// TIA Portal V19 export
DATA_BLOCK "Coilcar"   // DB112
// stored: InstanceOfName Coilcar_FB, InstanceOfType FB
"Coilcar_FB"
   // VAR_INPUT
   //    AreaInterface : "AreaInterface";
   //    ZSI : "udt_ZoneSafetyInterface";
   //    DSI : Struct
   //       Move : "udt_DeviceSafetyInterface";
   //       LIft : "udt_DeviceSafetyInterface";
   //    END_STRUCT;
   //    Drive : "TAx_DriveInterface";
   //    HW_ID_TEL1 : HW_SUBMODULE;
   //    DataIn : Struct
   //       Supports_Ls_FixPoleLeft_Plugged : Bool;
   //       Supports_Ls_FixPoleRight_Plugged : Bool;
   //       Supports_Ls_MobilePoleLeft_Plugged : Bool;
   //       Supports_Ls_MobilePoleRight_Plugged : Bool;
   //       Move_Ls_Outline : Bool;
   //       Move_Ls_Inline : Bool;
   //       Move_Ls_LowSpeedOutline : Bool;
   //       Move_Ls_LowSpeedInline : Bool;
   //       Move_Ls_CoilInserted : Bool;
   //       Move : "SpeedMachine_DataIn";
   //       Lift1 : "ValveMachine_DataIn";
   //       Lift2 : "ValveMachine_DataIn";
   //    END_STRUCT;
   //    CIn : Struct
   //       PressureRunning : Bool;
   //    END_STRUCT;
   //    Config : Struct
   //       LsStopDelayON { ExternalAccessible := 'False'; ExternalVisible := 'False'; ExternalWritable := 'False'} : Time;
   //       LsStopDelayOFF { ExternalAccessible := 'False'; ExternalVisible := 'False'; ExternalWritable := 'False'} : Time;
   //       Move : "SpeedMachine_Config";
   //       Lift1 : "ValveMachine_Config";
   //       Lift2 : "ValveMachine_Config";
   //    END_STRUCT;
   // END_VAR
   // VAR_OUTPUT
   //    MachineInterface : "MachineInterface";
   //    DataOut : Struct
   //       Move : "SpeedMachine_DataOut";
   //       Lift1 : "ValveMachine_DataOut";
   //       Lift2 : "ValveMachine_DataOut";
   //    END_STRUCT;
   //    COut : Struct
   //       IsInline : Bool;
   //       IsOutline : Bool;
   //       Move : "SpeedMachine_COut";
   //       Lift1 : "ValveMachine_COut";
   //       Lift2 : "ValveMachine_COut";
   //    END_STRUCT;
   // END_VAR
   // VAR_IN_OUT
   //    PersistentValues : Struct
   //       Move : "SpeedMachine_Par";
   //    END_STRUCT;
   // END_VAR
   // VAR
   //    Sts : Struct
   //       Move : Struct
   //          LowSpeedInline : Bool;
   //          LowSpeedOutline : Bool;
   //          IsInline : Bool;
   //          IsOutline : Bool;
   //          Inline_Cnd : Bool;
   //          Outline_Cnd : Bool;
   //          ReductionRatio : LReal;
   //       END_STRUCT;
   //       Free : Bool;
   //    END_STRUCT;
   //    Alarm : Struct
   //       Move_UnvalidStateLsInOut : Bool;
   //       Move_UnvalidStateLsLow : Bool;
   //       Move : "SpeedMachine_Alr";
   //       Lift1 : "ValveAlr";
   //       Lift2 : "ValveAlr";
   //    END_STRUCT;
   //    Warning : Struct
   //       Move : "SpeedMachine_Wng";
   //       Lift1 { ExternalAccessible := 'False'; ExternalVisible := 'False'; ExternalWritable := 'False'} : "ValveMachine_Wng";
   //       Lift2 { ExternalAccessible := 'False'; ExternalVisible := 'False'; ExternalWritable := 'False'} : "ValveMachine_Wng";
   //       NotOutline : Bool;
   //       Supports_FixPolesNotPlugged : Bool;
   //       Supports_MobilePolesNotPlugged : Bool;
   //    END_STRUCT;
   //    Move : "SpeedMachine_FB";
   //    Lift1 : "ValveMachine_FB";
   //    Lift2 : "ValveMachine_FB";
   //    TON_OutlinePos_DelayON : IEC_TIMER;
   //    TON_OutlinePos_DelayOFF : IEC_TIMER;
   //    TON_InlinePos_DelayON : IEC_TIMER;
   //    TON_InlinePos_DelayOFF : IEC_TIMER;
   //    pippo { S7_SetPoint := 'True'} : IEC_TIMER;
   // END_VAR
BEGIN
   AreaInterface.EStop := FALSE;
   AreaInterface.Man := TRUE;
   AreaInterface.Aut := FALSE;
   AreaInterface.Cycle := FALSE;
   AreaInterface.StopInPhase := FALSE;
   AreaInterface.StopProgrammed := FALSE;
   AreaInterface.RstAlarms := FALSE;
   AreaInterface.ManOneShot := FALSE;
   AreaInterface.AutOneShot := FALSE;
   AreaInterface.CycleOneShot := FALSE;
   AreaInterface.CheckAutReady := FALSE;
   MachineInterface.AutReady := FALSE;
   MachineInterface.Aborting := FALSE;
   MachineInterface.AckStopInPhase := FALSE;
   MachineInterface.AckStopProgrammed := FALSE;
   MachineInterface.MotionsStandStill := TRUE;
   MachineInterface.AlarmsPresence := FALSE;
   MachineInterface.WarningPresence := FALSE;
END_DATA_BLOCK
